(* CODESYS project library.library
   Company: Beckhoff Application
   DefaultNamespace: Tc3_TComObjectServer
   Version: 1.1.6
   Placeholder: Tc3_TComObjectServer
   Author: Beckhoff Application
   Description: Library to interact with the TwinCAT 3.1 TCom ObjectServer for handling and creating dynamic TCom Objects.
   Title: Tc3_TComObjectServer

Project tree, tasks and I/O mapping:
  libraries: Tc2_Standard, * (Beckhoff Automation GmbH); Tc2_System, * (Beckhoff Automation GmbH); Tc2_Utilities, * (Beckhoff Automation GmbH); Tc3_Module, * (Beckhoff Automation GmbH)
  [internal]/
    function DeleteTcBaseModule [ST]
    function PTComAdsCreateInstanceDATA [ST]
    function PTComInitDataElmSIZE [ST]
    data type TComAdsCreateInstance
    function block TComBaseModuleFactory [ST]
  DataTypes/
    data type ParameterInit
  Version/
    global variables Global_Version
  function DeleteTComObject [ST]
  function block TComGetModulesByClass [ST]
  function block TComModuleFactory [ST]: FB_exit
*)

// [internal]/TComAdsCreateInstance
{attribute {attribute 'pack_mode' := '1'}
{attribute 'hide'}
{attribute 'conditional_show'}
TYPE TComAdsCreateInstance :
STRUCT
  ClassID 				: GUID;
  ObjectID 				: OTCID;
  ParentObjectID 		: OTCID;
  TargetState 			: TCOM_STATE;
  {attribute 'hide'}
  _Reserved 			: ARRAY [0..4] OF UDINT;

  Name 					: STRING(127);
  ParameterInitSize 	: UDINT;
END_STRUCT
END_TYPE

// DataTypes/ParameterInit
TYPE
    ParameterInit :
    STRUCT
        PID  : PTCID;
        Data : PVOID;
        Size : UDINT;
    END_STRUCT
END_TYPE

// Version/Global_Version
{attribute 'TcGenerated'}
{attribute 'no-analysis'}
{attribute 'linkalways'}
// This function has been automatically generated from the project information.
VAR_GLOBAL CONSTANT
	{attribute 'const_non_replaced'}
	stLibVersion_Tc3_TComObjectServer : ST_LibVersion := (iMajor := 1, iMinor := 1, iBuild := 6, iRevision := 0, nFlags := 1, sVersion := '1.1.6');
END_VAR

// [internal]/DeleteTcBaseModule
{attribute 'hide'}
{attribute 'conditional_show'}
FUNCTION DeleteTcBaseModule : HRESULT
VAR_INPUT
    Module : REFERENCE TO Tc3_Module.TcBaseModule;
END_VAR
VAR
    _result : REFERENCE TO HRESULT;
END_VAR

_result REF= DeleteTcBaseModule;

IF NOT __ISVALIDREF(Module) THEN
    RETURN;
END_IF

_result := Module
    .TcSetObjState(TCOM_STATE.TCOM_STATE_SAFEOP, TwinCAT_SystemInfoVarList._AppInfo.TComSrvPtr, 0);

IF FAILED(_result) THEN
    RETURN;
END_IF

_result := Module
    .TcSetObjState(TCOM_STATE.TCOM_STATE_PREOP, TwinCAT_SystemInfoVarList._AppInfo.TComSrvPtr, 0);

IF FAILED(_result) THEN
    RETURN;
END_IF

_result := Module
    .TcSetObjState(TCOM_STATE.TCOM_STATE_INIT, TwinCAT_SystemInfoVarList._AppInfo.TComSrvPtr, 0);

IF FAILED(_result) THEN
    RETURN;
END_IF

_result := TO_DINT(Module.TcRelease());

IF FAILED(_result) THEN
    RETURN;
END_IF

END_FUNCTION

// [internal]/PTComAdsCreateInstanceDATA
{attribute 'hide'}
{attribute 'conditional_show'}
FUNCTION PTComAdsCreateInstanceDATA : POINTER TO Tc3_Module.TComInitDataHdr
VAR_INPUT
  p   : POINTER TO TComAdsCreateInstance;
END_VAR
VAR
END_VAR

PTComAdsCreateInstanceDATA := p + SIZEOF(TComAdsCreateInstance);

END_FUNCTION

// [internal]/PTComInitDataElmSIZE
{attribute 'hide'}
{attribute 'conditional_show'}
FUNCTION PTComInitDataElmSIZE : UDINT
VAR_INPUT
  n : UDINT;
END_VAR

PTComInitDataElmSIZE := (sizeof(TComInitDataElmHdr) + (n));

END_FUNCTION

// [internal]/TComBaseModuleFactory
{attribute 'hide'}
{attribute 'conditional_show'}
{attribute 'hide_all_locals'}
FUNCTION_BLOCK TComBaseModuleFactory
VAR_INPUT
    Execute : BOOL;
    Name : STRING(127);
    ObjectID : OTCID := Tc3_Module.OTCID_CreateNewId;
    ClassID : CLSID;
    Parent : OTCID := 16#00000000;
    TargetState : TCOM_STATE := TCOM_STATE.TCOM_STATE_OP;
END_VAR

VAR_IN_OUT
    ParameterInit : ARRAY[*] OF ParameterInit;
END_VAR

VAR_OUTPUT
    Busy : BOOL;
    Error : BOOL;
    ErrorID : UDINT;
    CreatedModule : POINTER TO Tc3_Module.TcBaseModuleRegistered;
END_VAR

VAR
    _moduleFactory : TComModuleFactory;
    _pBaseModule : POINTER TO Tc3_Module.TcBaseModuleRegistered;
END_VAR

_moduleFactory(
    Execute:=Execute,
    Name:=Name,
    ObjectID:=ObjectID,
    ClassID:=ClassID,
    Parent:=Parent,
    TargetState:=TargetState,
    ParameterInit:=ParameterInit,
    Busy=>Busy,
    Error=>Error,
    ErrorID=>ErrorID,
    CreatedObjectID=>
);

IF _moduleFactory.CreatedObjectID <> 0 AND NOT _moduleFactory.Busy THEN
    _pBaseModule := __NEW(Tc3_Module.TcBaseModuleRegistered(sObjectName:=Name));

    _pBaseModule^.TcSetObjectId(ObjectID);
    _pBaseModule^.TcSetObjectName(ADR(Name));
    _pBaseModule^.TcSetParentObjId(Parent);

    CreatedModule := _pBaseModule;
END_IF

END_FUNCTION_BLOCK

// TComModuleFactory
{attribute 'hide_all_locals'}
FUNCTION_BLOCK TComModuleFactory
VAR_INPUT
    Execute : BOOL;
    Name : STRING(127);
    ObjectID : OTCID := Tc3_Module.OTCID_CreateNewId; // [OPTIONAL]
    ClassID : CLSID; 
	Library : STRING := ''; // [OPTIONAL] e.g. C++ Module Vendor|MyModule|0.0.0.1
	TaskContext : OTCID := 16#0; // [OPTIONAL] e.g. object id of a cyclic task
    Parent : OTCID := 16#0; // [OPTIONAL]
    TargetState : TCOM_STATE := TCOM_STATE.TCOM_STATE_OP; // [OPTIONAL]
END_VAR

VAR_IN_OUT
    ParameterInit : ARRAY[*] OF ParameterInit; // [OPTIONAL]
END_VAR

VAR_OUTPUT
    Busy : BOOL;
    Error : BOOL;
    ErrorID : UDINT;
    CreatedObjectID : OTCID;
END_VAR

VAR
    _dataSize : UDINT;
    _dynamicData : POINTER TO BYTE;
    _objectID : OTCID;

    _createTComModule : Tc2_System.ADSRDWRT;

    _pCreateInstance : POINTER TO TComAdsCreateInstance;
    _pDataHeader : POINTER TO Tc3_Module.TComInitDataHdr;
    _pParameterInit : POINTER TO Tc3_Module.TComInitDataElmHdr;

    _onExecute : R_TRIG;
    _state : (
        IDLE,
        CREATE_MODULE,
        DONE,
        ERROR
    );
    i : DINT;

    _paramLowerBound : DINT;
    _paramUpperBound : DINT;

    _paramCount : DINT;

    _ipParentObject	: ITComObject;
    _doesParentExist : HRESULT;

    _ipComObject	: ITComObject;
    _doesObjectAlreadyExist : HRESULT;
	_classIdVersioned : CLSID;
	_isValidTaskObjectId : HRESULT;
	_ipTask : ITcTask;
	
	_taskPriority : UDINT;
	_taskCycleTimeNs : UDINT;
END_VAR

VAR CONSTANT
    TOMSERVER_ADS_PORT : T_AmsPort := 12;
    TCOMSERVER_IGRP_CREATEINSTANCE : UDINT := 16#00000003;
    EMPTY_CLASS_ID : CLSID := STRING_TO_GUID('00000000-0000-0000-0000-000000000000');
	
	PID_TASK_CONTEXT : PTCID := 16#03002060; // OTCID
	PID_TASK_PRIORITY : PTCID := 16#03002070; // UDINT
	PID_TASK_CYCLE_TIME_NS : PTCID := 16#3002080; // UDINT
	PID_TASK_PORT : PTCID := 16#03002090; // UINT
	PID_TASK_SORT_ORDER : PTCID := 16#030020B0; // UDINT
	PID_TRACE_LEVEL_MAX : PTCID := 16#00000001; // TcTraceLevel
END_VAR

_onExecute( CLK := Execute );

IF _onExecute.Q AND NOT Busy THEN

    _paramLowerBound := 0;
    _paramUpperBound := 0;
    _paramCount      := 0;

    CreatedObjectID := 0;
	Busy 			:= FALSE;
    Error           := FALSE;
    ErrorID         := 0;

    IF Name = '' THEN
        Error   := TRUE;
        ErrorID := E_AdsErr.DEVICE_INVALIDDATA;
        RETURN;
    END_IF

    IF GuidsEqual( ADR( ClassID ), ADR( EMPTY_CLASS_ID ) ) THEN
        Error   := TRUE;
        ErrorID := E_AdsErr.DEVICE_INVALIDCLSID;
        RETURN;
    END_IF

    IF Library <> '' THEN

        IF FIND( Library, '|' ) = 0 THEN // invalid library format
            Error   := TRUE;
            ErrorID := E_AdsErr.DEVICE_INVALIDCLSID;
            RETURN;
        END_IF

        IF NOT F_GetClassIdVersioned( Library, ClassID, _classIdVersioned ) THEN
            Error   := TRUE;
            ErrorID := E_AdsErr.DEVICE_INVALIDCLSID;
            RETURN;
        END_IF
    ELSE
        _classIdVersioned := ClassID;
    END_IF

    IF ObjectID <> Tc3_Module.OTCID_CreateNewId THEN
        FW_ObjMgr_GetObjectInstance( ObjectID, TC_GLOBAL_IID_LIST.IID_ITComObject, ADR( _ipComObject ) );

        IF _ipComObject <> 0 THEN
            Error   := TRUE;
            ErrorID := E_AdsErr.DEVICE_INVALIDOBJID;

            FW_SafeRelease( ADR( _ipComObject ) );
            RETURN;
        END_IF

        IF ObjectID < OTCID_FirstFreeId OR ObjectID > OTCID_LastFreeId THEN
            Error   := TRUE;
            ErrorID := E_AdsErr.DEVICE_INVALIDOBJID;
            RETURN;
        END_IF
    END_IF

    IF Parent <> 0 THEN
        _doesParentExist := FW_ObjMgr_GetObjectInstance( Parent, TC_GLOBAL_IID_LIST.IID_ITComObject, ADR( _ipParentObject ) );

        IF FAILED( _doesParentExist ) THEN
            Error   := TRUE;
            ErrorID := E_AdsErr.DEVICE_INVALIDOBJID;
            RETURN;
        ELSE
            FW_SafeRelease( ADR( _ipParentObject ) );
        END_IF
    END_IF

    IF ParameterInit <> 0 THEN
        _paramLowerBound := LOWER_BOUND( ParameterInit, 1 );
        _paramUpperBound := UPPER_BOUND( ParameterInit, 1 );

		_paramCount := _paramUpperBound - _paramLowerBound + 1;
    ELSE
        _paramCount := 0;
    END_IF

    _dataSize := SIZEOF( TComAdsCreateInstance );
	
	IF _paramCount > 0 OR TaskContext <> 16#0 THEN
		_dataSize := _dataSize + SIZEOF( TComInitDataHdr );
	END_IF

    IF _paramCount > 0 THEN

        FOR i := _paramLowerBound TO _paramUpperBound DO

            IF ParameterInit[i].PID = 16#0 THEN
                CONTINUE;
            END_IF

            IF ParameterInit[i].PID <> 16#0 AND (ParameterInit[i].Size = 0 OR ParameterInit[i].Data = 0)
                THEN
                Busy    := FALSE;
                Error   := TRUE;
                ErrorID := E_AdsErr.DEVICE_INVALIDDATA;
                RETURN;
            END_IF

            _dataSize := _dataSize + PTComInitDataElmSize( ParameterInit[i].Size );
        END_FOR

    END_IF

    IF TaskContext <> 16#0 THEN

        _isValidTaskObjectId := FW_ObjMgr_GetObjectInstance( TaskContext, TC_GLOBAL_IID_LIST.IID_ITcTask, ADR( _ipTask ) );

        IF FAILED( _isValidTaskObjectId ) THEN
            Error   := TRUE;
            ErrorID := E_AdsErr.DEVICE_INVALIDCONTEXT;
            RETURN;
        ELSE
			
			_ipTask.GetPriority(ADR(_taskPriority));
			_ipTask.GetCycleTime(ADR(_taskCycleTimeNs));

            FW_SafeRelease( ADR( _ipTask ) );
        END_IF

        _dataSize   := _dataSize + PTComInitDataElmSize( SIZEOF( OTCID ) ); // TASK CONTEXT
		_dataSize   := _dataSize + PTComInitDataElmSize( SIZEOF( UDINT ) ); // TASK PRIORITY
		_dataSize   := _dataSize + PTComInitDataElmSize( SIZEOF( UDINT ) ); // TASK CYCLE TIME NS
    END_IF

    IF _dynamicData <> 0 THEN
        __DELETE( _dynamicData );
    END_IF

    _dynamicData := __NEW( BYTE, _dataSize );

    IF _dynamicData = 0 THEN
        Error   := TRUE;
        ErrorID := E_AdsErr.DEVICE_NOMEMORY;
        RETURN;
    END_IF

    //MEMSET(_dynamicData, 0, _dataSize);

    _pCreateInstance := _dynamicData;

    _pCreateInstance^.ClassID           := _classIdVersioned;
    _pCreateInstance^.Name              := name;
    _pCreateInstance^.ObjectID          := ObjectID;
    _pCreateInstance^.ParentObjectID    := Parent;
    _pCreateInstance^.TargetState       := TargetState;
    _pCreateInstance^.ParameterInitSize := _dataSize - SIZEOF( TComAdsCreateInstance );

    IF _paramCount > 0 THEN

        _pDataHeader           := PTComAdsCreateInstanceDATA( _pCreateInstance );
        _pDataHeader^.uiElmCnt := 0;
        _pDataHeader^.cbData   := _pCreateInstance^.ParameterInitSize - SIZEOF( TComInitDataHdr );

        _pParameterInit := _pDataHeader;

        FOR i := _paramLowerBound TO _paramUpperBound DO

            IF ParameterInit[i].PID = 0 THEN
                CONTINUE;
            END_IF

            IF ParameterInit[i].Data <> 0 AND
               ParameterInit[i].Size > 0 AND
               ParameterInit[i].PID <> 0 THEN

                _pParameterInit              := Tc3_Module.PTComInitDataElmHdrNEXTHDR( _pParameterInit );
                _pParameterInit^.cbData      := ParameterInit[i].Size;
                _pParameterInit^.indexGroup  := 0;
                _pParameterInit^.indexOffset := ParameterInit[i].PID;

                MEMCPY(
                    Tc3_Module.PTComInitDataElmHdrDATA( _pParameterInit ),
                    ParameterInit[i].Data,
                    ParameterInit[i].Size
                );

                _pDataHeader^.uiElmCnt := _pDataHeader^.uiElmCnt + 1;

            END_IF
        END_FOR
    END_IF

    IF TaskContext <> 16#0 THEN
        IF _paramCount = 0 THEN
            _pDataHeader           := PTComAdsCreateInstanceDATA( _pCreateInstance );
            _pDataHeader^.uiElmCnt := 0;
            _pDataHeader^.cbData   := _pCreateInstance^.ParameterInitSize - SIZEOF( TComInitDataHdr );

            _pParameterInit := _pDataHeader;
        END_IF

		// Task Context
        _pParameterInit              := Tc3_Module.PTComInitDataElmHdrNEXTHDR( _pParameterInit );
        _pParameterInit^.cbData      := SIZEOF( OTCID );
        _pParameterInit^.indexGroup  := 0;
        _pParameterInit^.indexOffset := PID_TASK_CONTEXT;

        MEMCPY(
            Tc3_Module.PTComInitDataElmHdrDATA( _pParameterInit ),
            ADR( TaskContext ),
            SIZEOF( TaskContext )
        );

        _pDataHeader^.uiElmCnt := _pDataHeader^.uiElmCnt + 1;

		// Task Priority
        _pParameterInit              := Tc3_Module.PTComInitDataElmHdrNEXTHDR( _pParameterInit );
        _pParameterInit^.cbData      := SIZEOF( UDINT );
        _pParameterInit^.indexGroup  := 0;
        _pParameterInit^.indexOffset := PID_TASK_PRIORITY;

        MEMCPY(
            Tc3_Module.PTComInitDataElmHdrDATA( _pParameterInit ),
            ADR( _taskPriority ),
            SIZEOF( _taskPriority )
        );

        _pDataHeader^.uiElmCnt := _pDataHeader^.uiElmCnt + 1;
		
		// Task Cycle Time NS
        _pParameterInit              := Tc3_Module.PTComInitDataElmHdrNEXTHDR( _pParameterInit );
        _pParameterInit^.cbData      := SIZEOF( UDINT );
        _pParameterInit^.indexGroup  := 0;
        _pParameterInit^.indexOffset := PID_TASK_CYCLE_TIME_NS;

        MEMCPY(
            Tc3_Module.PTComInitDataElmHdrDATA( _pParameterInit ),
            ADR( _taskCycleTimeNs ),
            SIZEOF( _taskCycleTimeNs )
        );

        _pDataHeader^.uiElmCnt := _pDataHeader^.uiElmCnt + 1;
    END_IF

    Busy   := TRUE;
    _state := CREATE_MODULE;
END_IF

CASE _state OF

    IDLE:
		
		Busy := FALSE;
		
		IF NOT Execute THEN
			Error := FALSE;
			ErrorID := 0;
			CreatedObjectID := 0;
		END_IF

    CREATE_MODULE:

        _createTComModule(
            PORT     := TOMSERVER_ADS_PORT,
            IDXGRP   := TCOMSERVER_IGRP_CREATEINSTANCE,
            IDXOFFS  := 0,
            WRTRD    := TRUE,
            WRITELEN := _dataSize,
            SRCADDR  := _dynamicData,
            READLEN  := SIZEOF( _objectID ),
            DESTADDR := ADR( _objectID )
        );

        IF NOT _createTComModule.BUSY THEN
            IF NOT _createTComModule.ERR THEN
                _state          := DONE;
                CreatedObjectID := _objectID;
            ELSE
                ErrorID := _createTComModule.ERRID;
                _state  := ERROR;
            END_IF

            __DELETE( _dynamicData );
            _dynamicData := 0;

            _pCreateInstance := 0;
            _pDataHeader     := 0;
            _pParameterInit  := 0;

            _paramCount      := 0;
            _paramLowerBound := 0;
            _paramUpperBound := 0;

            _createTComModule( WRTRD := FALSE );
        END_IF

    DONE:
        Busy   := FALSE;
        _state := IDLE;

        IF ObjectID <> Tc3_Module.OTCID_CreateNewId THEN
            IF ObjectID <> CreatedObjectID THEN
                Error   := TRUE;
                ErrorID := E_AdsErr.DEVICE_INVALIDOBJID;
            END_IF
        END_IF

    ERROR:
        Busy   := FALSE;
        Error  := TRUE;
        _state := IDLE;

END_CASE

{attribute 'hide'}
METHOD FB_exit : BOOL
VAR_INPUT
    bInCopyCode : BOOL; // if TRUE, the exit method is called for exiting an instance that is copied afterwards (online change).
END_VAR
__DELETE(_dynamicData);

_dynamicData := 0;
_pCreateInstance := 0;
_pDataHeader := 0;
_pParameterInit := 0;

_paramCount := 0;
_paramLowerBound := 0;
_paramUpperBound := 0;
END_METHOD

END_FUNCTION_BLOCK

// DeleteTComObject
FUNCTION DeleteTComObject : HRESULT
VAR_INPUT
    ObjectID : OTCID;
END_VAR

VAR
    _ipComObject : ITComObject;
    _result      : HRESULT;
    _objectState : TCOM_STATE;
END_VAR

IF ObjectID = 0 THEN
    DeleteTComObject := E_HRESULTAdsErr.INVALIDDATA;
    RETURN;
END_IF

_result := Tc3_Module
    .FW_ObjMgr_GetObjectInstance( ObjectID, TC_GLOBAL_IID_LIST.IID_ITComObject, ADR( _ipComObject ) );

IF FAILED( _result ) OR _ipComObject = 0 THEN
	DeleteTComObject := _result;
    RETURN;
END_IF

_ipComObject.TcGetObjState( ADR( _objectState ) );

IF _objectState = TCOM_STATE.TCOM_STATE_OP THEN
    _result := _ipComObject
        .TcSetObjState( TCOM_STATE.TCOM_STATE_SAFEOP, TwinCAT_SystemInfoVarList._AppInfo.TComSrvPtr, 0 );

    IF FAILED( _result ) THEN
        DeleteTComObject := _result;
        RETURN;
    END_IF
END_IF

_ipComObject.TcGetObjState( ADR( _objectState ) );

IF _objectState = TCOM_STATE.TCOM_STATE_SAFEOP THEN
    _result := _ipComObject
        .TcSetObjState( TCOM_STATE.TCOM_STATE_PREOP, TwinCAT_SystemInfoVarList._AppInfo.TComSrvPtr, 0 );

    IF FAILED( _result ) THEN
        DeleteTComObject := _result;
        RETURN;
    END_IF
END_IF

_ipComObject.TcGetObjState( ADR( _objectState ) );

IF _objectState = TCOM_STATE.TCOM_STATE_PREOP THEN
    _result := _ipComObject
        .TcSetObjState( TCOM_STATE.TCOM_STATE_INIT, TwinCAT_SystemInfoVarList._AppInfo.TComSrvPtr, 0 );

    IF FAILED( _result ) THEN
        DeleteTComObject := _result;
        RETURN;
    END_IF
END_IF

_result := Tc3_Module.FW_ObjMgr_DeleteInstance( ADR( _ipComObject ) );

IF FAILED( _result ) THEN
    DeleteTComObject := _result;
    RETURN;
END_IF

_result := FW_SafeRelease( ADR( _ipComObject ) );

IF FAILED( _result ) THEN
    DeleteTComObject := _result;
    RETURN;
END_IF

_ipComObject := 0;

DeleteTComObject := _result;

END_FUNCTION

// TComGetModulesByClass
{attribute 'hide_all_locals'}
FUNCTION_BLOCK TComGetModulesByClass
VAR_INPUT
    Execute : BOOL;
    ClassID : CLSID;
    Library : STRING := ''; // [OPTIONAL] e.g. C++ Module Vendor|MyModule|0.0.0.1
END_VAR

VAR_IN_OUT
    ObjectIDs : ARRAY [*] OF OTCID;
END_VAR

VAR_OUTPUT
    Busy    : BOOL;
    Error   : BOOL;
    ErrorID : UDINT;
    Count   : UDINT;
END_VAR

VAR
    _onExecute          : R_TRIG;
    _getModuleObjectIDs : ADSRDWRT;

    _lowerBound : DINT;
    _upperBound : DINT;
    _dataSize   : UDINT;
    i           : DINT;
    _state      : (
        IDLE,
        EXEC,
        DONE,
        ERR
    );
    _classIdVersioned : CLSID;
END_VAR

VAR CONSTANT
    EMPTY_CLASS_ID : CLSID := STRING_TO_GUID( '00000000-0000-0000-0000-000000000000' );
	TCOM_OBJECT_SERVER_ADS_PORT : T_AmsPort := 10;
	GET_MODULES_INDEX_GROUP : UDINT := 16#201;
	GET_MODULES_INDEX_OfFSET : UDINT := 16#02;
END_VAR

_onExecute( CLK := Execute );

IF _onExecute.Q AND NOT Busy THEN
    Error   := FALSE;
    ErrorID := 0;
    Count   := 0;

    IF GuidsEqual( ADR( ClassID ), ADR( EMPTY_CLASS_ID ) ) THEN
        Error   := TRUE;
        ErrorID := E_AdsErr.DEVICE_INVALIDCLSID;
        RETURN;
    END_IF

    IF ObjectIDs = 0 THEN
        Error   := TRUE;
        ErrorID := E_AdsErr.DEVICE_INVALIDDATA;
        RETURN;
    END_IF

    _lowerBound := LOWER_BOUND( ObjectIDs, 1 );
    _upperBound := UPPER_BOUND( ObjectIDs, 1 );

    IF _lowerBound < 0 OR _upperBound < 0 THEN
        Error   := TRUE;
        ErrorID := E_AdsErr.DEVICE_INVALIDDATA;
        RETURN;
    END_IF

	_dataSize := TO_UDINT( _upperBound - _lowerBound + 1 );

    IF Library <> '' THEN
		
		IF FIND(Library, '|') = 0 THEN // invalid library format
			Error   := TRUE;
            ErrorID := E_AdsErr.DEVICE_INVALIDCLSID;
            RETURN;
		END_IF
	
        IF NOT F_GetClassIdVersioned( Library, ClassID, _classIdVersioned ) THEN
            Error   := TRUE;
            ErrorID := E_AdsErr.DEVICE_INVALIDCLSID;
            RETURN;
        END_IF
	ELSE
		_classIdVersioned := ClassID;
    END_IF

    Busy   := TRUE;
    _state := EXEC;

END_IF

CASE _state OF

    IDLE:
		Busy := FALSE;
		
		IF NOT Execute THEN
			Error := FALSE;
			ErrorID := 0;
			Count := 0;
		END_IF

    EXEC:

        _getModuleObjectIDs(
            NetID    := '',
            Port     := TCOM_OBJECT_SERVER_ADS_PORT,
            WRTRD    := TRUE,
            IDXGRP   := GET_MODULES_INDEX_GROUP,
            IDXOFFS  := GET_MODULES_INDEX_OfFSET,
            WRITELEN := SIZEOF( _classIdVersioned ),
            SRCADDR  := ADR( _classIdVersioned ),
            READLEN  := (_dataSize * SIZEOF( OTCID )),
            DESTADDR := ObjectIDs
        );

        IF NOT _getModuleObjectIDs.BUSY THEN
            IF NOT _getModuleObjectIDs.ERR THEN

                FOR i := _lowerBound TO _upperBound DO
                    IF ObjectIDs[i] <> 0 THEN
                        Count := Count + 1;
                    END_IF
                END_FOR

                _state := DONE;
            ELSE
                ErrorID := _getModuleObjectIDs.ERRID;
                _state  := ERR;
            END_IF

            _getModuleObjectIDs( WRTRD := FALSE );
        END_IF

    DONE:
        Busy   := FALSE;
        _state := IDLE;

    ERR:
        Error  := TRUE;
        Busy   := FALSE;
        _state := IDLE;

END_CASE

END_FUNCTION_BLOCK
